// TIA Portal V19 export
FUNCTION "B to b" : Void   // FC302, STL
TITLE = Convert Byte to bits
{ S7_Optimized_Access := 'TRUE' }
// stored: AutoNumber false
   VAR_INPUT
      iByte : Byte;
   END_VAR
   VAR_OUTPUT
      b_0 : Bool;
      b_1 : Bool;
      b_2 : Bool;
      b_3 : Bool;
      b_4 : Bool;
      b_5 : Bool;
      b_6 : Bool;
      b_7 : Bool;
   END_VAR
   VAR_TEMP
      iTmp : Byte;
   END_VAR
BEGIN

NETWORK
TITLE = 
      L     #iByte;
      T     #iTmp;

      A     #iTmp.%X0;
      =     #b_0;
      A     #iTmp.%X1;
      =     #b_1;
      A     #iTmp.%X2;
      =     #b_2;
      A     #iTmp.%X3;
      =     #b_3;
      A     #iTmp.%X4;
      =     #b_4;
      A     #iTmp.%X5;
      =     #b_5;
      A     #iTmp.%X6;
      =     #b_6;
      A     #iTmp.%X7;
      =     #b_7;





END_FUNCTION
